{attribute 'qualified_only'}
VAR_GLOBAL
	
	Input_Coils        	: ARRAY [0..255] OF BOOL;  	//R/W BOOLS
	Input_Registers     : ARRAY [0..255] OF WORD;	//R/W 16-Bit Register
	
	Output_Coils	    : ARRAY [0..255] OF BOOL;	//Read Only BOOLS
	Output_Registers    : ARRAY [0..255] OF WORD;	//Read Only 16-Bit Register
	
END_VAR

(*-----------------------------------------------------------------------------
Output_Coils[0]		- 1000 <- Licht Küche
Output_Coils[1] 	- 1001 <- Licht Hausgang EG
Output_Coils[2] 	- 1002 <- Aussenbeleuchtung OST 		
Output_Coils[3] 	- 1003 <- Aussenbeleuchtung Haustür 	
Output_Coils[4] 	- 1004 <- Licht Technikraum
Output_Coils[5] 	- 1005 <- Licht Hobbyraum
Output_Coils[6] 	- 1006 <- Licht Werkstatt
Output_Coils[7] 	- 1007 <- Licht Esszimmertisch
Output_Coils[8] 	- 1008 <- Licht Esszimmer
Output_Coils[9] 	- 1009 <- Licht Wohnzimmer
Output_Coils[10] 	- 1010 <- Aussenbeleuchtung Balkon
Output_Coils[11] 	- 1011 <- Wohnzimmer Steckdose Uhr
Output_Coils[12] 	- 1012 <- Werkstatt Steckdose
Output_Coils[13] 	- 1013 <- Garagentor Impuls
Output_Coils[14] 	- 1014 <- Türgong Impuls
Output_Coils[15] 	- 1015 <- Vitramo Bad
Output_Coils[16] 	- 1016 <- Haustüröffner Impuls
Output_Coils[17] 	- 1017 <- Haustüröffner Dauer
Output_Coils[18] 	- 1018 <- Wohnzimmer Steckdose Fernseher
Output_Coils[19] 	- 1019 <- ENV_NoDailight
Output_Coils[20] 	- 1020 <- Wohnzimmer Steckdose Esszimmer
Output_Coils[21] 	- 1021 <- Aussensteckdose Haustür
Output_Coils[22] 	- 1022 <- Aussensteckdose Balkon
Output_Coils[23] 	- 1023 <- Strom Zisternenpumpe
Output_Coils[24] 	- 1024 <- Strom SmartMirror
Output_Coils[25] 	- 1025 <- Wohnzimmer Steckdose LED-Band
Output_Coils[26] 	- 1026 <- Lüfter Werkstatt
Output_Coils[27] 	- 1027 <- Strom Heizung Werkstatt
Output_Coils[28] 	- 1028 <- 
Output_Coils[29] 	- 1029 <- 
Output_Coils[30] 	- 1030 <- 
Output_Coils[31] 	- 1031 <- 
Output_Coils[32] 	- 1032 <- 
Output_Coils[33] 	- 1033 <- 
Output_Coils[34] 	- 1034 <- 
Output_Coils[35] 	- 1035 <- 
Output_Coils[36] 	- 1036 <- 


########################----FENSTER / TÜRKONTAKTE----################
Output_coils[200]	- 1200 <- Fenster 	EG 	BAD
Output_coils[201]	- 1201 <- Fenster 	EG 	Büro
Output_coils[202]	- 1202 <- Tür		EG	Balkontür
Output_coils[203]	- 1203 <- Fenster	UG	Keller
Output_coils[204]	- 1204 <- Fenster	UG	Technik
Output_coils[205]	- 1205 <- Fenster	UG	Hobbyraum Süd
Output_coils[206]	- 1206 <- Fenster	UG	Hobbyraum West
Output_coils[207]	- 1207 <- Tür		UG	Terassentür
Output_coils[208]	- 1208 <- Fenster	UG	Werkstatt
Output_coils[209]	- 1209 <- Tür		UG	Werkstatt
Output_coils[210]	- 1210 <- 




########################----ALARM----################################
Output_coils[240]	- 1240 <- Aktiviert alle Alarmfunktionen

Output_coils[241]	- 1241 <- Aktiviert dauerhaft alle Lichter
Output_coils[242]	- 1242 <- Aktiviert dauerhaft alle Lichter INNEN
Output_coils[243]	- 1243 <- Aktiviert dauerhaft alle Lichter AUSSEN

Output_coils[244]	- 1244 <- Aktiviert dauerhaft alle Alarmsignale
Output_coils[245]	- 1245 <- Aktiviert dauerhaft alle Alarmsignale INNEN
Output_coils[246]	- 1246 <- Aktiviert dauerhaft alle Alarmsignale AUSSEN

Output_coils[247]	- 1247 <- 
Output_coils[248]	- 1248 <- 
Output_coils[249]	- 1249 <- 
Output_coils[250]	- 1250 <- 

Output_coils[251]	- 1251 <- Aktiviert Testalarm Esszimmertisch
Output_coils[252]	- 1252 <- Aktiviert Testalarm Esszimmer
Output_coils[253]	- 1253 <- Aktiviert Testalarm Wohnzimmer
Output_coils[254]	- 1254 <- Aktiviert Testalarm Balkon
Output_coils[255]	- 1255 <- 



------------------------------------------------------------------------------*)

(*-----------------------------------------------------------------------------
Output_Registers[0] 	- 2000 <- Trinkwasserverbrauch gvl_RETAIN 
Output_Registers[7] 	- 2007 <- Helligkeit Esszimmertisch
Output_Registers[8] 	- 2008 <- Helligkeit Esszimmer
Output_Registers[9] 	- 2009 <- Helligkeit Wohnzimmer
Output_Registers[10] 	- 2010 <- Helligkeit Aussenbeleuchtung Balkon
Output_Registers[11] 	- 2011 <- Zisterne Füllstand mA
Output_Registers[12] 	- 2012 <- Zisterne Füllstand Prozent
Output_Registers[13] 	- 2013 <- Zisterne Füllstand Liter
Output_Registers[14] 	- 2014 <- Wohnzimmer Temperatur
Output_Registers[15] 	- 2015 <- Wohnzimmer Feuchtigkeit
Output_Registers[16] 	- 2016 <- Wohnzimmer CO2
Output_Registers[17] 	- 2017 <- Technikraum Temperatur
Output_Registers[18] 	- 2018 <- Technikraum Feuchtigkeit
Output_Registers[19] 	- 2019 <- Dachboden Temperatur
Output_Registers[20] 	- 2020 <- Werkstatt Temperatur
Output_Registers[21] 	- 2021 <- Werkstatt Feuchtigkeit
Output_Registers[22] 	- 2022 <- 



------------------------------------------------------------------------------*)

(* stored: Version 1.1.0.1, ProductVersion 3.1.4024.4
   GVL gvl_mb: Id {3db55538-7040-430d-8b30-7a8f8b1e24d7} *)
